TYPE "LubrValve_HMI"
VERSION : 0.1
// Block: LubrValve_HMI
   STRUCT
      ManReq : Bool;
      AutoReq : Bool;
      Running : Bool;
      Alarm : Bool;
      ActualWorkTime : Time;
   END_STRUCT;

END_TYPE
